FUNCTION_BLOCK Test_AddEventHandler_IncsNumberOfEventHandlers EXTENDS TUnitTestbase
VAR_INPUT
END_VAR
VAR_OUTPUT
END_VAR
VAR
    TestEvent : TTestEvent;
    TestEventHandler : TTestEventHandler;
END_VAR

METHOD  Execute
Test_Started();

TestEvent
    .ClearEventHandlers()
    .AddEventHandler(TestEventHandler);
    
Assertion.AssertEquals_UDINT(
    Expected := 1,
    Actual   := TestEvent.EventHandlers.Count,
    ObjectName := _TestName,
    VariableName  := 'TestEvent.EventHandlers.Count');
    

Test_Finished();
END_METHOD

END_FUNCTION_BLOCK

(* stored: Version 1.1.0.1, ProductVersion 3.1.4024.3
   POU Test_AddEventHandler_IncsNumberOfEventHandlers: Id {eda56f75-f01d-4e29-8f23-82687b9fbdd7}, SpecialFunc None
   Method Execute: Id {ee8a7f4a-6051-4ab5-8403-72f2bd5fec94} *)
